INTERFACE I_DataChannelSend

PROPERTY Busy : BOOL
GET
END_GET
END_PROPERTY

{attribute 'object_name' := 'ClearBufferDone'}
METHOD ClearBufferDone : BOOL
END_METHOD

{attribute 'object_name' := 'SendData'}
METHOD SendData : BOOL
VAR_INPUT
	udiDataSize: UDINT;
	pData: POINTER TO BYTE;
END_VAR
END_METHOD

PROPERTY DataSize : UDINT
GET
END_GET
END_PROPERTY

PROPERTY Error : INT
GET
END_GET
SET
END_SET
END_PROPERTY

PROPERTY ClearBufferRequest : BOOL
GET
END_GET
END_PROPERTY

{attribute 'object_name' := 'InitChannel'}
METHOD InitChannel : BOOL
VAR_INPUT
	udiDataSize: UDINT;
	pOutputData: POINTER TO BYTE;
END_VAR
END_METHOD

END_INTERFACE

(* stored: Version 1.1.0.1, ProductVersion 3.1.0.26
   Itf I_DataChannelSend: Id {75d65f29-9061-4ec0-98e9-366b36792db5}
   Property Busy: Id {09072595-833a-4ce3-b03f-a7e253820814}
   Get Get: Id {c427a56a-b079-494b-bdb5-35d154fca078}
   Method ClearBufferDone: Id {6b5a9877-63cd-4bdd-a676-ba741a8b6165}
   Method SendData: Id {925bea83-f2ed-4f5f-824b-f4ac3008a371}
   Property DataSize: Id {a9f62bac-efc6-4071-a51e-1c21b5e51419}
   Get Get: Id {d6d8af02-791a-40ea-b813-e02cdb7dc4e9}
   Property Error: Id {b8738404-b2fe-4754-a6d8-d590e53cadce}
   Get Get: Id {d20bdfe6-2260-4145-a6ef-bff27968ad00}
   Set Set: Id {d5711c38-aefc-4a81-82e4-4284e9e31535}
   Property ClearBufferRequest: Id {c93a6dac-5ea8-4430-9e37-ff9ddeb2a588}
   Get Get: Id {803dc20c-6312-4af6-9d74-2254fd6fecbb}
   Method InitChannel: Id {ea2c8c13-35a8-4402-9028-818467207db1} *)
